(* CoDeSys 2.3.9.41 project: press_7.pro *)
(* Libraries: STANDARD.LIB 4.10.05 11:14:46, IECSFC.LIB 13.4.06 15:51:28, ANALYZATION.LIB 5.10.99 09:05:06, D:\Sespel\Стенды\Пресс\Прорамма\ПЛК100\SysLibTime.lib 17.10.19 08:53:27 *)

(* PLC configuration (modules and I/O channels)
Discrete input 8 bit [ID100] node 0, in %IB0 out %QB0 {Filtrationtime = 10; Filtrationtime = 10; Filtrationtime = 10; Filtrationtime = 10; Filtrationtime = 10; Filtrationtime = 10; Filtrationtime = 10; Filtrationtime = 10; Visibility = No; PinCount = 8; WatchDogPeriod = 1000; PollPeriod = 1}
  AT %IB0.0 [ByteInput] 8 discrete inputs
Discrete output - relay [ID102] node 1, in %IB1 out %QB1 {PinCount = 1; SafeValueBool = FALSE; Visibility = No}
  AT %QX1.0 [BitOutput] relay
Discrete output - relay [ID102] node 2, in %IB2 out %QB2 {PinCount = 1; SafeValueBool = FALSE; Visibility = No}
  AT %QX2.0 [BitOutput] relay
Discrete output - relay [ID102] node 3, in %IB3 out %QB3 {PinCount = 1; SafeValueBool = FALSE; Visibility = No}
  AT %QX3.0 [BitOutput] relay
Discrete output - relay [ID102] node 4, in %IB4 out %QB4 {PinCount = 1; SafeValueBool = FALSE; Visibility = No}
  AT %QX4.0 [BitOutput] relay
Discrete output - relay [ID102] node 5, in %IB5 out %QB5 {PinCount = 1; SafeValueBool = FALSE; Visibility = No}
  AT %QX5.0 [BitOutput] relay
Discrete output - relay [ID102] node 6, in %IB6 out %QB6 {PinCount = 1; SafeValueBool = FALSE; Visibility = No}
  AT %QX6.0 [BitOutput] relay
Special output [ID104] node 7, in %IB7 out %QB7 {Visibility = No; PinCount = 1}
  AT %QX7.0 [BitOutput] Special output
AT %QD8.0 [DWordOutput] Last address
AT %QW8.1 [WordOutput] Last error
RS-485-1 [COM1_USART] node 0, in %IB8.0 out %QB8.0 {CommunicationSpeed = 57600; Parity = NO PARITY CHECK; BitLength = 8 bits; StopLength = One stop bit; InterfaceType = RS485; FrameOriented = RTU; Timeout = 0; Visibility = No}
AT %QB8.1.0 [ComChannel] Command (0xff - Start)
pr200_dd AT %IW8.1.0.0 [WordInput]
pr200_dd_zad AT %IW8.1.1.0 [WordInput]
pr200_YP AT %IW8.1.2.0 [WordInput]
ModBus (slave) [MODBUS_ID400] node 9, in %IB9 out %QB9 {SlaveIdentificator = 1; Visibility = No}
Cloud [TCP_ID222] node 0, in %IB9.0.0 out %QB9.0.0 {RemotePort = 25502; CloudServerIPFileName = owencloud.txt; CloudToken = MUWOGMWZ; Visibility = No}
cloud_dd AT %QD9.1.0 [FloatOutput]
cloud_YP AT %QW9.2.0 [WordOutput]
cloud_dd_zad AT %QD9.3.0 [FloatOutput]
cloud_zagruzka AT %QD9.4.0 [FloatOutput]
TCP [TCP_ID221] node 0, in %IB10.0.0 out %QB10.0.0 {RemotePort = 502; Visibility = No}
tcp_dd AT %QD10.1.0 [FloatOutput]
tcp_YP AT %QW10.2.0 [WordOutput]
tcp_dd_zad AT %QD10.3.0 [FloatOutput]
tcp_zagruzka AT %QD10.4.0 [FloatOutput]
tcp_chas AT %QW10.5.0 [WordOutput]
tcp_min AT %QW10.6.0 [WordOutput]
tcp_sec AT %QW10.7.0 [WordOutput]
tcp_tok_a AT %QW10.8.0 [WordOutput]
tcp_tok_b AT %QW10.9.0 [WordOutput]
tcp_tok_c AT %QW10.10.0 [WordOutput]
Button [ID003] node 11, in %IB11 out %QB11
  AT %IX11.0 [BitInput] Button Start/Stop
AT %QD12.0 [DWordOutput] Last address
AT %QW12.1 [WordOutput] Last error
RS-485-1 [COM1_USART] node 0, in %IB12.0 out %QB12.0 {CommunicationSpeed = 11520; Parity = NO PARITY CHECK; BitLength = 8 bits; StopLength = One stop bit; InterfaceType = RS485; FrameOriented = ASCII; Timeout = 0; Visibility = No}
AT %QB12.1.0 [ComChannel] Command (0xff - Start)
tcp595_tok_a AT %IW12.1.0.0 [WordInput]
tcp595_tok_b AT %IW12.1.1.0 [WordInput]
tcp595_tok_c AT %IW12.1.2.0 [WordInput]
*)

(* POU PLC_PRG, ST *)
PROGRAM PLC_PRG
VAR RETAIN
	GetTime: CurTimeEx;
	TimeAndDate: SystemTimeDate;
	Sys_Time: SysTime64;
	set_time: BOOL;
	set_date: BOOL;
	MM: UINT;
	SS: UINT;
	HH: UINT;
	D: UINT;
	M: UINT;
	Y: UINT;

	t1:TON;
	t1_trig:R_TRIG;
	t1_in: BOOL;
      t1_real:REAL;
	t1_time:TIME;
	sec: WORD;
	minut:WORD;

	prostoi: REAL;
	zagruzka_sutki:REAL;
	zagruzka_okrugl:REAL;
END_VAR
VAR

END_VAR
(*Owencloud*)
cloud_dd:=pr200_dd*0.0084;
cloud_YP:=pr200_YP;
cloud_dd_zad:=pr200_dd_zad*0.1;
cloud_zagruzka:=zagruzka_okrugl;

(*Умный дом*)
tcp_dd:=cloud_dd;
tcp_YP:=cloud_YP;
tcp_dd_zad:=cloud_dd_zad;
tcp_zagruzka:=cloud_zagruzka;
tcp_chas:=TimeAndDate.Hour;
tcp_min:=TimeAndDate.Minute;
tcp_sec:=TimeAndDate.Second;

(*Текущее время*)
TimeAndDate.Day :=0;
TimeAndDate.DayOfWeek :=0;
TimeAndDate.dwHighMsec :=0;
TimeAndDate.dwLowMSecs :=0;
TimeAndDate.Milliseconds :=0;
TimeAndDate.Minute :=0;
TimeAndDate.Second :=0;
TimeAndDate.Hour :=0;
TimeAndDate.Year :=0;
TimeAndDate.Month :=0;
Sys_time.ulHigh :=0;
Sys_time.ulLow :=0;
GetTime (SystemTime:=Sys_Time , TimeDate:= TimeAndDate);

(*Если set_time - истина, то можно менять время*)
IF set_time THEN
	TimeAndDate.Minute:= 42;
	TimeAndDate.Second:=0;
	TimeAndDate.Hour:=9;
	GetTime (SystemTime:=Sys_Time , TimeDate:= TimeAndDate);
END_IF

(*Обнуляем время по окончанию суток*)
IF TimeAndDate.Hour=0 AND TimeAndDate.Minute =0 AND TimeAndDate.Second =0 THEN
sec:=0;
END_IF

(*Счетчик загруженности за сутки*)
zagruzka_sutki:=sec/864.00;
zagruzka_okrugl:=DINT_TO_REAL(REAL_TO_DINT(zagruzka_sutki*100))/100; (*для огругления до двух знаков после запятой*)
prostoi:=100-zagruzka_okrugl;

(*Таймер с 1 секундным счетчиком*)
IF pr200_YP=1 THEN
t1_time:=WORD_TO_TIME(1000); (*Преобразовываем значение 1 секунда*)
t1(IN:=t1_in,PT:=t1_time);   (*Запускаем таймер *)
t1_trig(CLK:=t1.Q);
t1_in:=TRUE;
END_IF

IF t1_trig.Q  THEN
sec:=sec+1;
t1_in:=FALSE;
END_IF

(*Отправляем показания тока с Индукционной печи*)
END_PROGRAM
